{attribute 'linkalways'}
{attribute 'hide_all_locals'}
FUNCTION_BLOCK ValueSint EXTENDS ValueSintRead IMPLEMENTS Value
VAR
END_VAR

METHOD SetFromType : BOOL
VAR_INPUT
	source : __SYSTEM.AnyType;
END_VAR
SetFromType := ConvertAnyType(source, thisAnyType);
END_METHOD

METHOD SetFromString : BOOL
VAR_INPUT
	value : T_MaxString;
END_VAR
thisValue := STRING_TO_SINT(value);

SetFromString := TRUE;
END_METHOD

METHOD Set : BOOL
VAR_INPUT
	source : ANY;
END_VAR
Set := ConvertAnyType(source, thisAnyType);
END_METHOD

END_FUNCTION_BLOCK

(* stored: Version 1.1.0.1
   POU ValueSint: Id {77f87b5c-cde0-4e66-89ee-c3f98a93ef2f}, SpecialFunc None
   Method SetFromType: Id {01d1452f-4bdb-4c55-b2c8-11e4c611b565}
   Method SetFromString: Id {fe050438-110b-44f9-9f56-76244a55369a}
   Method Set: Id {d2614c14-6b47-4e87-bd59-1f0b9c12a3a7} *)
